FUNCTION_BLOCK InitializableComponent_Mockup EXTENDS CyclicComponent IMPLEMENTS I_Initializable
VAR
	_Initialized		 : BOOL;
	_WasCalled			 : BOOL;
	_InitializeWasCalled : BOOL;
END_VAR

METHOD CyclicLogic
_WasCalled := TRUE;
END_METHOD

METHOD Initialize
_InitializeWasCalled := TRUE;
END_METHOD

{attribute 'monitoring' := 'call'}
PROPERTY Initialized : BOOL
GET
Initialized := _Initialized;
END_GET
SET
_Initialized := Initialized;
END_SET
END_PROPERTY

PROPERTY InitializeWasCalled : BOOL
GET
InitializeWasCalled := _InitializeWasCalled;
END_GET
END_PROPERTY

PROPERTY WasCalled : BOOL
GET
WasCalled := _WasCalled;
END_GET
END_PROPERTY

END_FUNCTION_BLOCK

(* stored: Version 1.1.0.1, ProductVersion 3.1.4026.18
   POU InitializableComponent_Mockup: Id {0237d679-3fbe-430d-ab9d-4b5eace52461}, SpecialFunc None
   Method CyclicLogic: Id {e17420a8-da52-4418-a33e-8a620976bf99}
   Method Initialize: Id {ea814110-96a1-4b70-be99-de90aab3cac0}
   Property Initialized: Id {659c2ca7-5371-45b7-8a37-97a800f80ce9}
   Get Get: Id {0d59e794-595c-4564-bcc3-3b6c39e07e8a}
   Set Set: Id {75b7efef-09c4-4669-9af2-37eb657b7bed}
   Property InitializeWasCalled: Id {0ce6dcf3-3f21-4912-9b52-248db5b25acb}
   Get Get: Id {ad23f689-a61a-40ae-b413-959f283e2896}
   Property WasCalled: Id {34d7e35b-df19-429e-b4a5-2c9fc9b2f868}
   Get Get: Id {f6135d86-2384-4926-9c68-f5e1d3003fe0} *)
